FUNCTION_BLOCK CU00xAutomat EXTENDS TcoTaskedSequencer IMPLEMENTS ICUTask
VAR
END_VAR

Run();

(*~
	<docu>
		<summary>
			Main method of the sequener. Custom code needs to be placed here. The sequencer is executed by call of **Instance.Run()** method.
			This method is abstract, and it must be overridden in derived block.
		</summary>
	</docu>
~*)
METHOD PROTECTED Main : BOOL
IF (Step(100, TRUE, 'LOAD PROCESS SETTING')) THEN
    //-------------------------------------
    Station.ProcessDataManager.Data := Station.Technology.ProcessSettings.Data;
	CompleteStep();
    //-------------------------------------
END_IF

IF (Step(200, TRUE, 'SINGLE INSPECTION')) THEN
    //-------------------------------------    
	Station.ProcessDataManager.Data.CU00x.BoltPresenceInspector
					.WithCoordinator(THIS^)
					.Inspect(FALSE)
					.UpdateComprehensiveResult(Station.ProcessDataManager.Data._entityHeader.Results)
					.OnFail().Dialog(100);	
    //-------------------------------------
END_IF

IF (Step(RESTORE_STEP_ID, TRUE, 'FIRST RESTORE STEP')) THEN
    //-------------------------------------
    StepCompleteWhen(%MX0.0);
    //-------------------------------------	
END_IF

IF (Step(10000, TRUE, 'LAST STEP')) THEN
    //-------------------------------------
    CompleteSequence();
    //-------------------------------------	
END_IF
END_METHOD

METHOD PUBLIC OnStart
Station.Ground.Restore();
Station.Manual.Restore();
END_METHOD

PROPERTY Station : REFERENCE TO CU00x
GET
VAR
    _station : POINTER TO CU00x;
END_VAR
IF __QUERYPOINTER(Parent, _station) THEN // Check if _Parent is Station001
    Station REF= _station^;              // If the check is successful dereference a pointer. simlar to THIS^ or SUPER^
END_IF
END_GET
END_PROPERTY

END_FUNCTION_BLOCK

(* stored: Version 1.1.0.1, ProductVersion 3.1.4024.9
   POU CU00xAutomat: Id {7d4ccf14-fbfb-4c7b-8fab-cda3fabc0370}, SpecialFunc None
   Method Main: Id {65c64653-c354-4e9f-878f-19a4b135c641}
   Method OnStart: Id {8fe4788f-029c-4df9-a93a-9297bee7e169}
   Property Station: Id {2f34bbe0-ae77-4424-96f8-d75571b12d83}
   Get Get: Id {5ff633c4-e770-483e-b525-87fa0c0de322} *)
